Staubli VAL3: new.pgx

public program new(trsf& x_tTool[])
  local num l_nSize
  local tool l_tTool
begin
  // only fifo politic
  call getSize(l_nSize)
  // TRSF
  insert(saveData:tData[l_nSize])
  l_tTool.trsf=x_tTool
  call setTool(l_tTool,l_nSize)
end
